// TIA Portal V19 export
FUNCTION_BLOCK "A0302_HU_Cytropack_FB"   // FB16, LAD
// stored: MemoryReserve 100, SetENOAutomatically false
   VAR_INPUT
      AreaInterface : "AreaInterface";
      ZSI : "udt_ZoneSafetyInterface";
      DSI : "udt_DeviceSafetyInterface";
      DataIn : Struct
         Pb_Stop : Bool;
         Pb_Start : Bool;
      END_STRUCT;
      CIn : Struct
         Manager : Struct
            EnableStopDoorOpeningReq { ExternalWritable := 'False'} : Bool;
            EnableStopInPhase { ExternalWritable := 'False'} : Bool;
            EnableStopProgrammed { ExternalWritable := 'False'} : Bool;
            Control_ON { ExternalWritable := 'False'} : Bool;
            Rest { ExternalWritable := 'False'} : Bool;
            Work { ExternalWritable := 'False'} : Bool;
         END_STRUCT;
         SemiAut_Pb { ExternalAccessible := 'False'; ExternalVisible := 'False'; ExternalWritable := 'False'} : Bool;
         PressureReq : Bool;
         PressureRunning : Bool;
         CarroPareggTesta : Struct
            Bloccaggio { ExternalAccessible := 'False'; ExternalVisible := 'False'; ExternalWritable := 'False'} : "ValveMachine_COut";
         END_STRUCT;
         CarroPareggCoda : Struct
            Bloccaggio { ExternalAccessible := 'False'; ExternalVisible := 'False'; ExternalWritable := 'False'} : "ValveMachine_COut";
            PareggiatoreLong { ExternalAccessible := 'False'; ExternalVisible := 'False'; ExternalWritable := 'False'} : "ValveMachine_COut";
         END_STRUCT;
      END_STRUCT;
      InputADDR : HW_IO := 16#0;   // Input address of the drive in hardware configuration
      OutputADDR : HW_IO := 16#0;   // Output address of the drive in hardware configuration
   END_VAR
   VAR_OUTPUT
      MachineInterface : "MachineInterface";
      COut : Struct
         Standstill : Bool;
         Run_CheckNext : Bool;
         CtrlSafe : Bool;
         PressureRunning : Bool;
         PressureInTarget : Bool;
      END_STRUCT;
   END_VAR
   VAR_IN_OUT
      Par : Struct
         Bloccaggio : Struct
            TargetPressure : Real;
            TargetSpeed : Real;
            Delta : Struct
               Min : Real;
               Max : Real;
            END_STRUCT;
         END_STRUCT;
         Pareggiamento : Struct
            TargetPressure : Real;
            TargetSpeed : Real;
            Delta : Struct
               Min : Real;
               Max : Real;
            END_STRUCT;
         END_STRUCT;
      END_STRUCT;
   END_VAR
   VAR
      M_Chiller : "Motor";
      Sts : Struct
         Standstill : Bool;
         AlarmsPresence : Bool;
         WarningsPresence : Bool;
         Cnd : Bool;
      END_STRUCT;
      Ctrl : Struct
         StopDueDoorOpeningRequest : Bool;
         StopInPhase : Bool;
         StopProgrammed : Bool;
         StopAborting : Bool;
         Run : Bool;
         Run_Man : Bool;
         Run_Aut : Bool;
      END_STRUCT;
      Alarm : Struct
         M_Chiller { S7_SetPoint := 'True'} : "MotorAlr";
         Fc_P5020 : Struct
            Error { S7_SetPoint := 'True'} : Bool;
            Warning : Bool;
         END_STRUCT;
         Fc_Diagn : Struct
            "0" : Bool;
            "1" : Bool;
            "2" : Bool;
            "3" : Bool;
            "4" : Bool;
            "5" : Bool;
            "6" : Bool;
            "7" : Bool;
            "8" : Bool;
            "9" : Bool;
            "10" : Bool;
            "11" : Bool;
            "12" : Bool;
            "13" : Bool;
            "14" : Bool;
            "15" : Bool;
         END_STRUCT;
      END_STRUCT;
      Warning : Struct
         NotAutReady : Bool;
      END_STRUCT;
      TON_NoPendingCmd : IEC_TIMER;
      TON_Inactivity : IEC_TIMER;
      TON_Pressure { S7_SetPoint := 'True'} : IEC_TIMER;
      Aux : Struct
         Pb_Start : Bool;
         ReqParBloccaggio : Bool;
         ReqParParegg : Bool;
      END_STRUCT;
   END_VAR
   VAR DB_SPECIFIC
      iReturnVal : Int := 0;   // Return value variable
      Error : Bool := false;   // Error active on the EFC / FcP function / function block
      bFBErrorDPRD_DPWR : Bool := false;   // Internal flag
      stInputData { S7_SetPoint := 'True'} : "FCP_IN";   // Input data structure
      stOutputData { S7_SetPoint := 'True'} : "FCP_OUT";   // Output data structure
   END_VAR
   VAR
      Range_TargetBlocc : Struct
         Min : Real;
         Max : Real;
      END_STRUCT;
      Range_TargetParegg : Struct
         Min : Real;
         Max : Real;
      END_STRUCT;
      Target : Struct
         Pressure_Value { ExternalAccessible := 'False'; ExternalVisible := 'False'; ExternalWritable := 'False'} : Real;
         MaxSpeed_Value { ExternalAccessible := 'False'; ExternalVisible := 'False'; ExternalWritable := 'False'} : Real;
      END_STRUCT;
   END_VAR
   VAR_TEMP
      PE : Struct
         OP_Rest_PB : Bool;
         OP_Work_PB : Bool;
      END_STRUCT;
   END_VAR
   VAR_TEMP   // added for the SCL form of the ladder/FBD networks
      _w1 : Bool;
      _w2 : Bool;
   END_VAR
BEGIN

REGION Network 1: << HU Bosch Rexroth>>
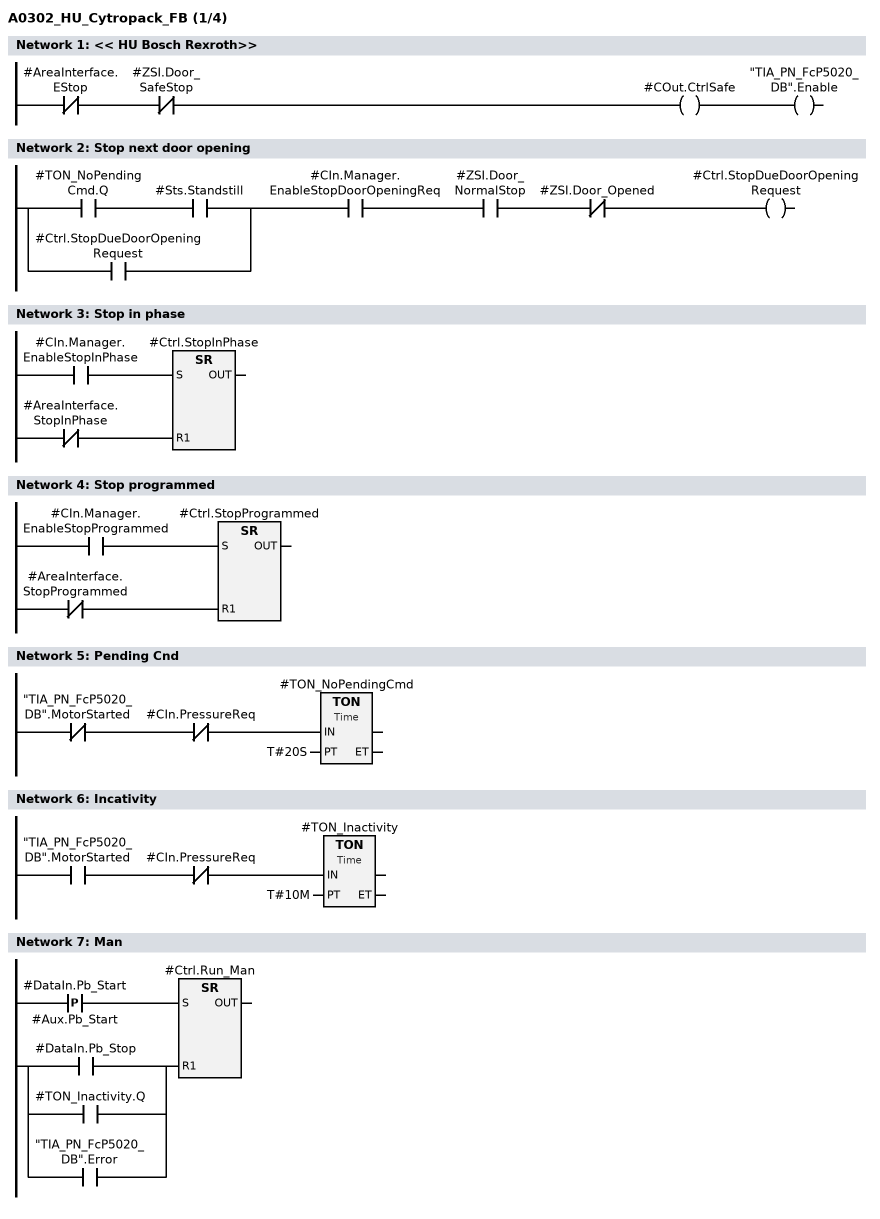
   RUNG wire#powerrail
      I_Contact( #AreaInterface.EStop )
      I_Contact( #ZSI.Door_SafeStop )
      Coil( #COut.CtrlSafe )
      Coil( "TIA_PN_FcP5020_DB".Enable )
   END_RUNG
   // the same network as SCL:
   #COut.CtrlSafe := NOT #AreaInterface.EStop AND NOT #ZSI.Door_SafeStop;
   "TIA_PN_FcP5020_DB".Enable := #COut.CtrlSafe;
END_REGION

REGION Network 2: Stop next door opening
   RUNG wire#powerrail
      Contact( #TON_NoPendingCmd.Q )
      Contact( #Sts.Standstill )
      wire#w1
      Contact( #CIn.Manager.EnableStopDoorOpeningReq )
      Contact( #ZSI.Door_NormalStop )
      I_Contact( #ZSI.Door_Opened )
      Coil( #Ctrl.StopDueDoorOpeningRequest )
   END_RUNG
   RUNG wire#powerrail
      Contact( #Ctrl.StopDueDoorOpeningRequest )
   END_RUNG wire#w1
   // the same network as SCL:
   #Ctrl.StopDueDoorOpeningRequest := ((#TON_NoPendingCmd.Q AND #Sts.Standstill) OR #Ctrl.StopDueDoorOpeningRequest) AND #CIn.Manager.EnableStopDoorOpeningReq AND #ZSI.Door_NormalStop AND NOT #ZSI.Door_Opened;
END_REGION

REGION Network 3: Stop in phase
   RUNG wire#powerrail
      Contact( #CIn.Manager.EnableStopInPhase )
      S_SR(operand := #Ctrl.StopInPhase, r1 := wire#w1)
   END_RUNG
   RUNG wire#powerrail
      I_Contact( #AreaInterface.StopInPhase )
   END_RUNG wire#w1
   // the same network as SCL:
   IF #CIn.Manager.EnableStopInPhase THEN
       #Ctrl.StopInPhase := TRUE;   // SR flip-flop
   END_IF;
   IF NOT #AreaInterface.StopInPhase THEN #Ctrl.StopInPhase := FALSE; END_IF;
END_REGION

REGION Network 4: Stop programmed
   RUNG wire#powerrail
      Contact( #CIn.Manager.EnableStopProgrammed )
      S_SR(operand := #Ctrl.StopProgrammed, r1 := wire#w1)
   END_RUNG
   RUNG wire#powerrail
      I_Contact( #AreaInterface.StopProgrammed )
   END_RUNG wire#w1
   // the same network as SCL:
   IF #CIn.Manager.EnableStopProgrammed THEN
       #Ctrl.StopProgrammed := TRUE;   // SR flip-flop
   END_IF;
   IF NOT #AreaInterface.StopProgrammed THEN #Ctrl.StopProgrammed := FALSE; END_IF;
END_REGION

REGION Network 5: Pending Cnd
   RUNG wire#powerrail
      I_Contact( "TIA_PN_FcP5020_DB".MotorStarted )
      I_Contact( #CIn.PressureReq )
      { S7_Templates := "time_type := Time" } #TON_NoPendingCmd.TON(pt := T#20S, et =>)
   END_RUNG
   // the same network as SCL:
   #TON_NoPendingCmd.TON(IN := NOT "TIA_PN_FcP5020_DB".MotorStarted AND NOT #CIn.PressureReq, PT := T#20S);
END_REGION

REGION Network 6: Incativity
   RUNG wire#powerrail
      Contact( "TIA_PN_FcP5020_DB".MotorStarted )
      I_Contact( #CIn.PressureReq )
      { S7_Templates := "time_type := Time" } #TON_Inactivity.TON(pt := T#10M, et =>)
   END_RUNG
   // the same network as SCL:
   #TON_Inactivity.TON(IN := "TIA_PN_FcP5020_DB".MotorStarted AND NOT #CIn.PressureReq, PT := T#10M);
END_REGION

REGION Network 7: Man
   RUNG wire#powerrail
      P_Contact(operand := #DataIn.Pb_Start, bit := #Aux.Pb_Start)
      S_SR(operand := #Ctrl.Run_Man, r1 := wire#w1)
   END_RUNG
   RUNG wire#powerrail
      Contact( #DataIn.Pb_Stop )
   END_RUNG wire#w1
   RUNG wire#powerrail
      Contact( #TON_Inactivity.Q )
   END_RUNG wire#w1
   RUNG wire#powerrail
      Contact( "TIA_PN_FcP5020_DB".Error )
   END_RUNG wire#w1
   // the same network as SCL:
   #_w1 := #DataIn.Pb_Start AND NOT #Aux.Pb_Start;   // rising edge of #DataIn.Pb_Start
   #Aux.Pb_Start := #DataIn.Pb_Start;
   IF #_w1 THEN
       #Ctrl.Run_Man := TRUE;   // SR flip-flop
   END_IF;
   IF #DataIn.Pb_Stop OR #TON_Inactivity.Q OR "TIA_PN_FcP5020_DB".Error THEN #Ctrl.Run_Man := FALSE; END_IF;
END_REGION

REGION Network 8: Aut
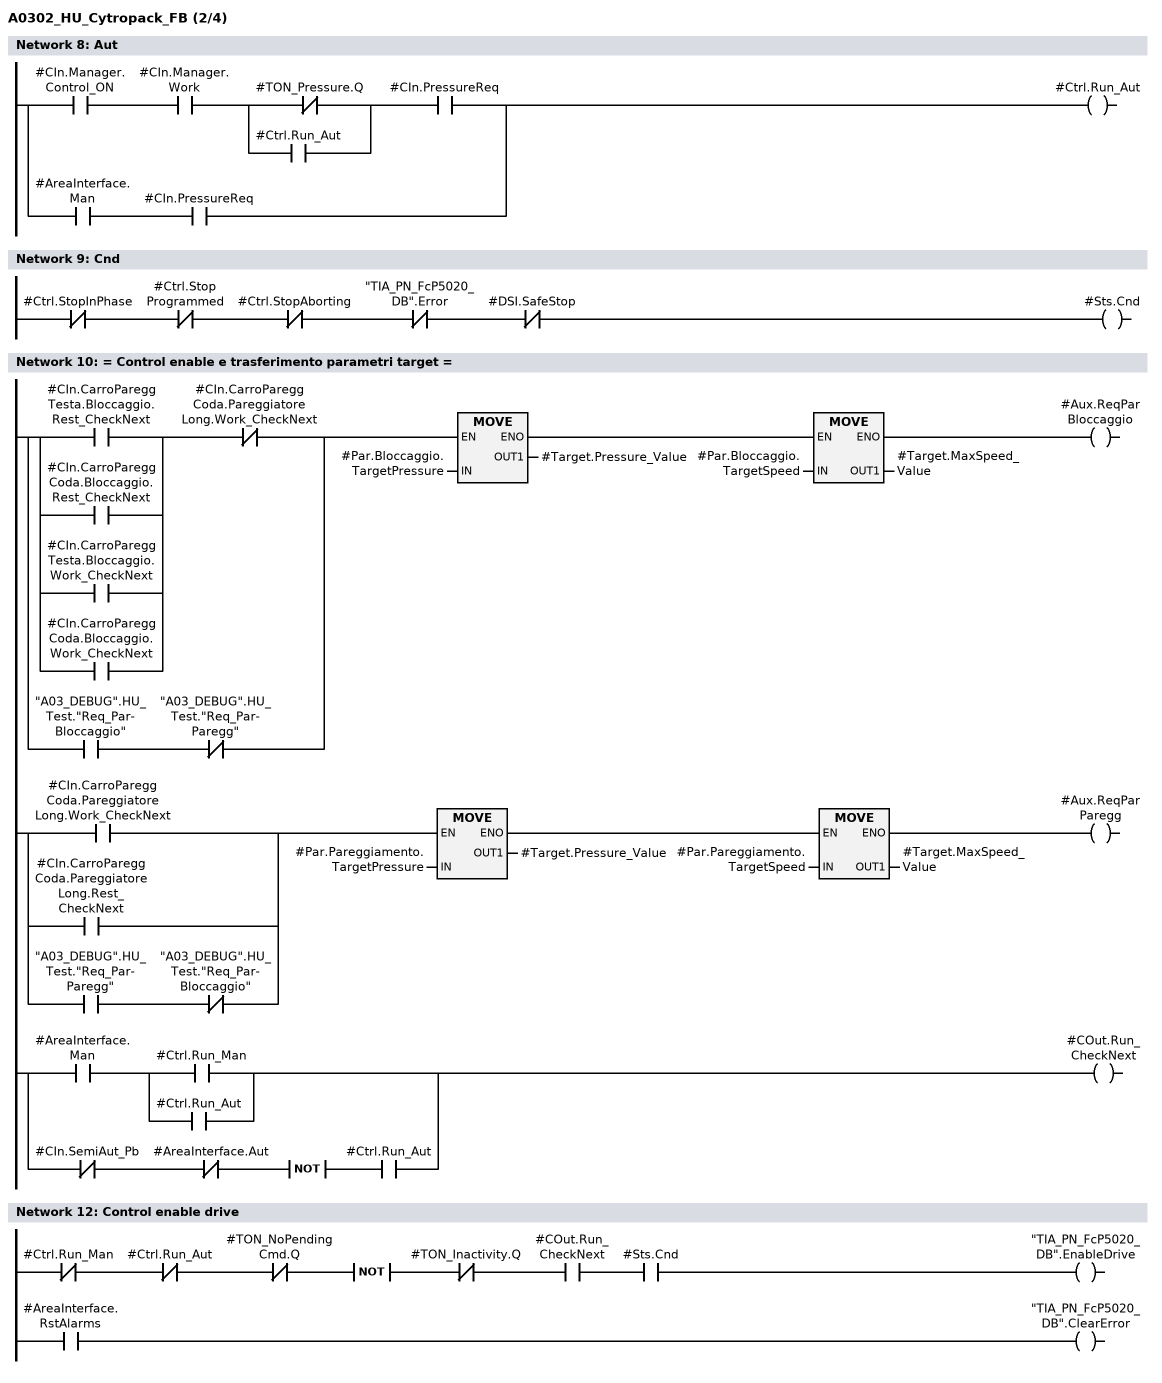
   RUNG wire#powerrail
      Contact( #CIn.Manager.Control_ON )
      Contact( #CIn.Manager.Work )
      wire#w1
      I_Contact( #TON_Pressure.Q )
      wire#w2
      Contact( #CIn.PressureReq )
      wire#w3
      Coil( #Ctrl.Run_Aut )
   END_RUNG
   RUNG wire#w1
      Contact( #Ctrl.Run_Aut )
   END_RUNG wire#w2
   RUNG wire#powerrail
      Contact( #AreaInterface.Man )
      Contact( #CIn.PressureReq )
   END_RUNG wire#w3
   // the same network as SCL:
   #Ctrl.Run_Aut := (#CIn.Manager.Control_ON AND #CIn.Manager.Work AND (NOT #TON_Pressure.Q OR #Ctrl.Run_Aut) AND #CIn.PressureReq) OR (#AreaInterface.Man AND #CIn.PressureReq);
END_REGION

REGION Network 9: Cnd
   RUNG wire#powerrail
      I_Contact( #Ctrl.StopInPhase )
      I_Contact( #Ctrl.StopProgrammed )
      I_Contact( #Ctrl.StopAborting )
      I_Contact( "TIA_PN_FcP5020_DB".Error )
      I_Contact( #DSI.SafeStop )
      Coil( #Sts.Cnd )
   END_RUNG
   // the same network as SCL:
   #Sts.Cnd := NOT #Ctrl.StopInPhase AND NOT #Ctrl.StopProgrammed AND NOT #Ctrl.StopAborting AND NOT "TIA_PN_FcP5020_DB".Error AND NOT #DSI.SafeStop;
END_REGION

REGION Network 10: = Control enable e trasferimento parametri target =
   RUNG wire#powerrail
      Contact( #CIn.CarroPareggTesta.Bloccaggio.Rest_CheckNext )
      wire#w1
      I_Contact( #CIn.CarroPareggCoda.PareggiatoreLong.Work_CheckNext )
      wire#w2
      Move(in := #Par.Bloccaggio.TargetPressure, out1 => #Target.Pressure_Value)
      Move(in := #Par.Bloccaggio.TargetSpeed, out1 => #Target.MaxSpeed_Value)
      Coil( #Aux.ReqParBloccaggio )
   END_RUNG
   RUNG wire#powerrail
      Contact( #CIn.CarroPareggCoda.Bloccaggio.Rest_CheckNext )
   END_RUNG wire#w1
   RUNG wire#powerrail
      Contact( #CIn.CarroPareggTesta.Bloccaggio.Work_CheckNext )
   END_RUNG wire#w1
   RUNG wire#powerrail
      Contact( #CIn.CarroPareggCoda.Bloccaggio.Work_CheckNext )
   END_RUNG wire#w1
   RUNG wire#powerrail
      Contact( "A03_DEBUG".HU_Test."Req_Par-Bloccaggio" )
      I_Contact( "A03_DEBUG".HU_Test."Req_Par-Paregg" )
   END_RUNG wire#w2
   RUNG wire#powerrail
      Contact( #CIn.CarroPareggCoda.PareggiatoreLong.Work_CheckNext )
      wire#w3
      Move(in := #Par.Pareggiamento.TargetPressure, out1 => #Target.Pressure_Value)
      Move(in := #Par.Pareggiamento.TargetSpeed, out1 => #Target.MaxSpeed_Value)
      Coil( #Aux.ReqParParegg )
   END_RUNG
   RUNG wire#powerrail
      Contact( #CIn.CarroPareggCoda.PareggiatoreLong.Rest_CheckNext )
   END_RUNG wire#w3
   RUNG wire#powerrail
      Contact( "A03_DEBUG".HU_Test."Req_Par-Paregg" )
      I_Contact( "A03_DEBUG".HU_Test."Req_Par-Bloccaggio" )
   END_RUNG wire#w3
   RUNG wire#powerrail
      Contact( #AreaInterface.Man )
      wire#w4
      Contact( #Ctrl.Run_Man )
      wire#w5
      Coil( #COut.Run_CheckNext )
   END_RUNG
   RUNG wire#w4
      Contact( #Ctrl.Run_Aut )
   END_RUNG wire#w5
   RUNG wire#powerrail
      I_Contact( #CIn.SemiAut_Pb )
      I_Contact( #AreaInterface.Aut )
      Not()
      Contact( #Ctrl.Run_Aut )
   END_RUNG wire#w5
   // the same network as SCL:
   #_w1 := ((#CIn.CarroPareggTesta.Bloccaggio.Rest_CheckNext OR #CIn.CarroPareggCoda.Bloccaggio.Rest_CheckNext OR #CIn.CarroPareggTesta.Bloccaggio.Work_CheckNext OR #CIn.CarroPareggCoda.Bloccaggio.Work_CheckNext) AND NOT #CIn.CarroPareggCoda.PareggiatoreLong.Work_CheckNext) OR ("A03_DEBUG".HU_Test."Req_Par-Bloccaggio" AND NOT "A03_DEBUG".HU_Test."Req_Par-Paregg");
   IF #_w1 THEN
       #Target.Pressure_Value := #Par.Bloccaggio.TargetPressure;
       #Target.MaxSpeed_Value := #Par.Bloccaggio.TargetSpeed;
   END_IF;
   #Aux.ReqParBloccaggio := #_w1;
   #_w2 := #CIn.CarroPareggCoda.PareggiatoreLong.Work_CheckNext OR #CIn.CarroPareggCoda.PareggiatoreLong.Rest_CheckNext OR ("A03_DEBUG".HU_Test."Req_Par-Paregg" AND NOT "A03_DEBUG".HU_Test."Req_Par-Bloccaggio");
   IF #_w2 THEN
       #Target.Pressure_Value := #Par.Pareggiamento.TargetPressure;
       #Target.MaxSpeed_Value := #Par.Pareggiamento.TargetSpeed;
   END_IF;
   #Aux.ReqParParegg := #_w2;
   #COut.Run_CheckNext := (#AreaInterface.Man AND (#Ctrl.Run_Man OR #Ctrl.Run_Aut)) OR (NOT (NOT #CIn.SemiAut_Pb AND NOT #AreaInterface.Aut) AND #Ctrl.Run_Aut);
END_REGION

REGION Network 11 (SCL): = Limiti sul target controllo pressione richiesta =
   // Limiti controllo Target Richiesta Bloccaggio
   #Range_TargetBlocc.Min := #Par.Bloccaggio.TargetPressure - #Par.Bloccaggio.Delta.Min;
   #Range_TargetBlocc.Max := #Par.Bloccaggio.TargetPressure + #Par.Bloccaggio.Delta.Max;

   // Limiti controllo Target Richiesta Pareggiamento Long
   #Range_TargetParegg.Min := #Par.Pareggiamento.TargetPressure - #Par.Pareggiamento.Delta.Min;
   #Range_TargetParegg.Max := #Par.Pareggiamento.TargetPressure + #Par.Pareggiamento.Delta.Max;
END_REGION

REGION Network 12: Control enable drive
   RUNG wire#powerrail
      I_Contact( #Ctrl.Run_Man )
      I_Contact( #Ctrl.Run_Aut )
      I_Contact( #TON_NoPendingCmd.Q )
      Not()
      I_Contact( #TON_Inactivity.Q )
      Contact( #COut.Run_CheckNext )
      Contact( #Sts.Cnd )
      Coil( "TIA_PN_FcP5020_DB".EnableDrive )
   END_RUNG
   RUNG wire#powerrail
      Contact( #AreaInterface.RstAlarms )
      Coil( "TIA_PN_FcP5020_DB".ClearError )
   END_RUNG
   // the same network as SCL:
   "TIA_PN_FcP5020_DB".EnableDrive := NOT (NOT #Ctrl.Run_Man AND NOT #Ctrl.Run_Aut AND NOT #TON_NoPendingCmd.Q) AND NOT #TON_Inactivity.Q AND #COut.Run_CheckNext AND #Sts.Cnd;
   "TIA_PN_FcP5020_DB".ClearError := #AreaInterface.RstAlarms;
END_REGION

REGION Network 13: Check Pressure
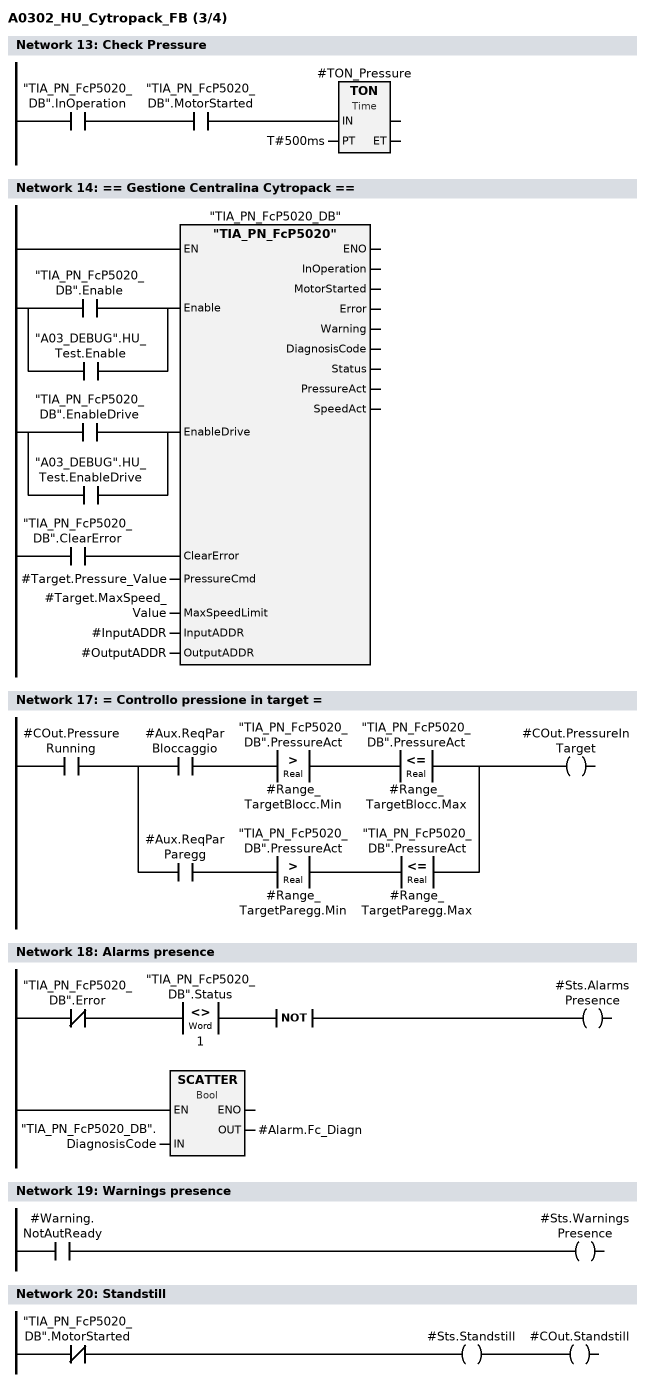
   RUNG wire#powerrail
      Contact( "TIA_PN_FcP5020_DB".InOperation )
      Contact( "TIA_PN_FcP5020_DB".MotorStarted )
      { S7_Templates := "time_type := Time" } #TON_Pressure.TON(pt := T#500ms, et =>)
   END_RUNG
   // the same network as SCL:
   #TON_Pressure.TON(IN := "TIA_PN_FcP5020_DB".InOperation AND "TIA_PN_FcP5020_DB".MotorStarted, PT := T#500ms);
END_REGION

REGION Network 14: == Gestione Centralina Cytropack ==
   RUNG wire#powerrail
      "TIA_PN_FcP5020_DB"(Enable := wire#w1, EnableDrive := wire#w2, ClearError := wire#w3, PressureCmd := #Target.Pressure_Value, MaxSpeedLimit := #Target.MaxSpeed_Value, InputADDR := #InputADDR, OutputADDR := #OutputADDR, InOperation =>, MotorStarted =>, Error =>, Warning =>, DiagnosisCode =>, Status =>, PressureAct =>, SpeedAct =>)
   END_RUNG
   RUNG wire#powerrail
      Contact( "TIA_PN_FcP5020_DB".Enable )
   END_RUNG wire#w1
   RUNG wire#powerrail
      Contact( "A03_DEBUG".HU_Test.Enable )
   END_RUNG wire#w1
   RUNG wire#powerrail
      Contact( "TIA_PN_FcP5020_DB".EnableDrive )
   END_RUNG wire#w2
   RUNG wire#powerrail
      Contact( "A03_DEBUG".HU_Test.EnableDrive )
   END_RUNG wire#w2
   RUNG wire#powerrail
      Contact( "TIA_PN_FcP5020_DB".ClearError )
   END_RUNG wire#w3
   // the same network as SCL:
   "TIA_PN_FcP5020_DB"(Enable := "TIA_PN_FcP5020_DB".Enable OR "A03_DEBUG".HU_Test.Enable,   // "TIA_PN_FcP5020"
                       EnableDrive := "TIA_PN_FcP5020_DB".EnableDrive OR "A03_DEBUG".HU_Test.EnableDrive,
                       ClearError := "TIA_PN_FcP5020_DB".ClearError,
                       PressureCmd := #Target.Pressure_Value,
                       MaxSpeedLimit := #Target.MaxSpeed_Value,
                       InputADDR := #InputADDR,
                       OutputADDR := #OutputADDR);
END_REGION

REGION Network 16: <<< MACHINE STATUS >>>
END_REGION

REGION Network 17: = Controllo pressione in target =
   RUNG wire#powerrail
      Contact( #COut.PressureRunning )
      wire#w1
      Contact( #Aux.ReqParBloccaggio )
      { S7_Templates := "SrcType := Real" } GT_Contact(in1 := "TIA_PN_FcP5020_DB".PressureAct, in2 := #Range_TargetBlocc.Min)
      { S7_Templates := "SrcType := Real" } LE_Contact(in1 := "TIA_PN_FcP5020_DB".PressureAct, in2 := #Range_TargetBlocc.Max)
      wire#w2
      Coil( #COut.PressureInTarget )
   END_RUNG
   RUNG wire#w1
      Contact( #Aux.ReqParParegg )
      { S7_Templates := "SrcType := Real" } GT_Contact(in1 := "TIA_PN_FcP5020_DB".PressureAct, in2 := #Range_TargetParegg.Min)
      { S7_Templates := "SrcType := Real" } LE_Contact(in1 := "TIA_PN_FcP5020_DB".PressureAct, in2 := #Range_TargetParegg.Max)
   END_RUNG wire#w2
   // the same network as SCL:
   #COut.PressureInTarget := #COut.PressureRunning AND ((#Aux.ReqParBloccaggio AND ("TIA_PN_FcP5020_DB".PressureAct > #Range_TargetBlocc.Min) AND ("TIA_PN_FcP5020_DB".PressureAct <= #Range_TargetBlocc.Max)) OR (#Aux.ReqParParegg AND ("TIA_PN_FcP5020_DB".PressureAct > #Range_TargetParegg.Min) AND ("TIA_PN_FcP5020_DB".PressureAct <= #Range_TargetParegg.Max)));
END_REGION

REGION Network 18: Alarms presence
   RUNG wire#powerrail
      I_Contact( "TIA_PN_FcP5020_DB".Error )
      { S7_Templates := "SrcType := Word" } NE_Contact(in1 := "TIA_PN_FcP5020_DB".Status, in2 := 1)
      Not()
      Coil( #Sts.AlarmsPresence )
   END_RUNG
   RUNG wire#powerrail
      { S7_Templates := "[dest_type := Bool, src_type := Word]" } SCATTER(IN := "TIA_PN_FcP5020_DB".DiagnosisCode, OUT => #Alarm.Fc_Diagn)
   END_RUNG
   // the same network as SCL:
   #Sts.AlarmsPresence := NOT (NOT "TIA_PN_FcP5020_DB".Error AND ("TIA_PN_FcP5020_DB".Status <> 1));
   SCATTER(IN := "TIA_PN_FcP5020_DB".DiagnosisCode, OUT => #Alarm.Fc_Diagn);
END_REGION

REGION Network 19: Warnings presence
   RUNG wire#powerrail
      Contact( #Warning.NotAutReady )
      Coil( #Sts.WarningsPresence )
   END_RUNG
   // the same network as SCL:
   #Sts.WarningsPresence := #Warning.NotAutReady;
END_REGION

REGION Network 20: Standstill
   RUNG wire#powerrail
      I_Contact( "TIA_PN_FcP5020_DB".MotorStarted )
      Coil( #Sts.Standstill )
      Coil( #COut.Standstill )
   END_RUNG
   // the same network as SCL:
   #Sts.Standstill := NOT "TIA_PN_FcP5020_DB".MotorStarted;
   #COut.Standstill := NOT "TIA_PN_FcP5020_DB".MotorStarted;
END_REGION

REGION Network 21: Stop for aborting
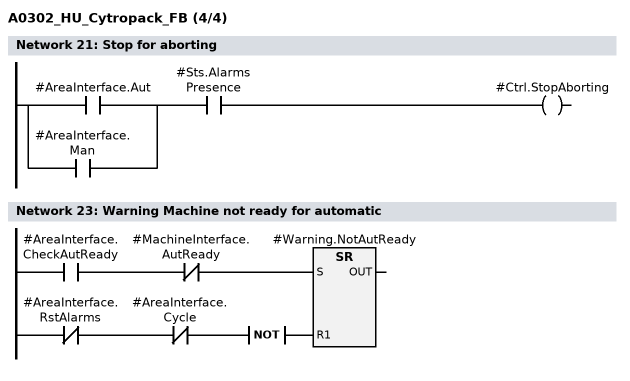
   RUNG wire#powerrail
      Contact( #AreaInterface.Aut )
      wire#w1
      Contact( #Sts.AlarmsPresence )
      Coil( #Ctrl.StopAborting )
   END_RUNG
   RUNG wire#powerrail
      Contact( #AreaInterface.Man )
   END_RUNG wire#w1
   // the same network as SCL:
   #Ctrl.StopAborting := (#AreaInterface.Aut OR #AreaInterface.Man) AND #Sts.AlarmsPresence;
END_REGION

REGION Network 22 (SCL): Collect machine to zone interface

   #MachineInterface.AutReady := #AreaInterface.Aut AND NOT #Sts.AlarmsPresence;
   #MachineInterface.Aborting := #Ctrl.StopAborting;
   #MachineInterface.MotionsStandStill := #TON_NoPendingCmd.Q AND #Sts.Standstill;
   #MachineInterface.AckStopInPhase := #Ctrl.StopInPhase  AND #MachineInterface.MotionsStandStill;
   #MachineInterface.AckStopProgrammed := #Ctrl.StopProgrammed AND #MachineInterface.MotionsStandStill;
   #MachineInterface.AlarmsPresence := #Sts.AlarmsPresence;
   #MachineInterface.WarningPresence := #Sts.WarningsPresence;
END_REGION

REGION Network 23: Warning Machine not ready for automatic
   RUNG wire#powerrail
      Contact( #AreaInterface.CheckAutReady )
      I_Contact( #MachineInterface.AutReady )
      S_SR(operand := #Warning.NotAutReady, r1 := wire#w1)
   END_RUNG
   RUNG wire#powerrail
      I_Contact( #AreaInterface.RstAlarms )
      I_Contact( #AreaInterface.Cycle )
      Not()
   END_RUNG wire#w1
   // the same network as SCL:
   IF #AreaInterface.CheckAutReady AND NOT #MachineInterface.AutReady THEN
       #Warning.NotAutReady := TRUE;   // SR flip-flop
   END_IF;
   IF NOT (NOT #AreaInterface.RstAlarms AND NOT #AreaInterface.Cycle) THEN
       #Warning.NotAutReady := FALSE;
   END_IF;
END_REGION

REGION Network 24 (SCL): Return value variable
   (* LBO TEST
   // Read data from EFC's PROFINET input area
   #iReturnVal := DPRD_DAT(LADDR := #InputADDR, RECORD => #stInputData);
   // Read data failed
   IF (#iReturnVal <> 0) THEN
       #Error := TRUE;
       #bFBErrorDPRD_DPWR := TRUE;
       RETURN;
   END_IF;
   *)
END_REGION
END_FUNCTION_BLOCK
